// TIA Portal V16 export
// export: Created 2024-09-05T17:39:24.390676Z, ExportSetting WithDefaults, DisplayName Totally Integrated Automation Portal, DisplayVersion V16 Update 6, DisplayName TIA Portal Version Control Interface, DisplayVersion V16 Update 2, DisplayName TIA Portal Openness, DisplayVersion V16 Update 6, DisplayName STEP 7 Professional, DisplayVersion V16 Update 6, DisplayName STEP 7 Safety, DisplayVersion V16, DisplayName WinCC Advanced, DisplayVersion V16 Update 6
FUNCTION_BLOCK "7. Call_M103_PY"   // FB2007, LAD
{ S7_Optimized_Access := 'TRUE' }
AUTHOR : bartz
VERSION : 0.1
// stored: AutoNumber false, IsIECCheckEnabled false, IsRetainMemResEnabled false, MemoryReserve 100, SetENOAutomatically false, UDAEnableTagReadback false
   VAR_INPUT
      PY_ON : Bool;
      PY_DOWN : Bool;
      PY_OFF : Bool;
   END_VAR
   VAR
      PYOnTemp : Bool;
      PYDownTemp : Bool;
      PYOffTemp : Bool;
   END_VAR
BEGIN

REGION Network 1 (SCL)
   IF (#PY_ON <> #PYOnTemp OR #PY_DOWN <> #PYDownTemp OR #PY_OFF <> #PYOffTemp) AND (#PY_ON OR #PY_DOWN OR #PY_OFF) THEN

       "MII_Interface_Data".MII_METHODS.M103_PY.Inputs.PLC_ID := "MII_Parameters".Connection.PLC_ID;
       "MII_Interface_Data".MII_METHODS.M103_PY.Inputs.PLANT := "MII_Parameters".Connection.PlantID;

       "MII_Interface_Data".MII_METHODS.M103_PY.Inputs.PY_ON := #PY_ON;
       "MII_Interface_Data".MII_METHODS.M103_PY.Inputs.PY_DOWN := #PY_DOWN;
       "MII_Interface_Data".MII_METHODS.M103_PY.Inputs.PY_OFF := #PY_OFF;

       //Call the method 
       "1. DMC_setConnection_DB".CallBuffer[7] := TRUE;

       #PYOnTemp := #PY_ON;
       #PYDownTemp := #PY_DOWN;
       #PYOffTemp := #PY_OFF;
   END_IF;
END_REGION
END_FUNCTION_BLOCK
